KUKA KRL program: chk_w2_grp3_opn.src, chk_w2_grp3_opn.dat

--- chk_w2_grp3_opn.src ---
&ACCESS RV2
&REL 3
&COMMENT Check grampos Z3 abertos
&PARAM DISKPATH = Program/SubeRotine
&PARAM TEMPLATE = C:\KRC\Roboter\Template\vorgabe
&PARAM EDITMASK = *
DEF chk_w2_grp3_opn( )
;FOLD ; Programa de verificacao de grampos Z3 aberto;%{PE}%R 4.1.16,%MKUKATPBASIS,%CCOMMENT,%VNORMAL,%P 2:Programa de verificacao de grampos Z3 aberto
;ENDFOLD

$TIMER[10] = 0
$TIMER_STOP[10] = FALSE

;FOLD WAIT FOR ( IN 499 'Z1.1 ABERTO/ ACTROS Z3.1 OPN' );%{PE}%R 8.2.24,%MKUKATPBASIS,%CEXT_WAIT_FOR,%VEXT_WAIT_FOR,%P 2:, 4:, 5:$IN, 6:499, 7:Z1.1 ABERTO/ ACTROS Z3.1 OPN, 9:
WAIT FOR  ( $IN[499] )
;ENDFOLD
;FOLD WAIT FOR ( IN 505 'ACTROS Z3.2 OPN' );%{PE}%R 8.2.24,%MKUKATPBASIS,%CEXT_WAIT_FOR,%VEXT_WAIT_FOR,%P 2:, 4:, 5:$IN, 6:505, 7:ACTROS Z3.2 OPN, 9:
WAIT FOR  ( $IN[505] )
;ENDFOLD
;FOLD WAIT FOR ( IN 507 'ACTROS 3.3 OPN' );%{PE}%R 8.2.24,%MKUKATPBASIS,%CEXT_WAIT_FOR,%VEXT_WAIT_FOR,%P 2:, 4:, 5:$IN, 6:507, 7:ACTROS 3.3 OPN, 9:
WAIT FOR  ( $IN[507] )
;ENDFOLD
;FOLD WAIT FOR ( IN 509 'ACTROS 3.4 OPN' );%{PE}%R 8.2.24,%MKUKATPBASIS,%CEXT_WAIT_FOR,%VEXT_WAIT_FOR,%P 2:, 4:, 5:$IN, 6:509, 7:ACTROS 3.4 OPN, 9:
WAIT FOR  ( $IN[509] )
;ENDFOLD
;FOLD WAIT FOR ( IN 513 'Z3.2 ABERTO/ ACTROS Z3.5 OPN' );%{PE}%R 8.2.24,%MKUKATPBASIS,%CEXT_WAIT_FOR,%VEXT_WAIT_FOR,%P 2:, 4:, 5:$IN, 6:513, 7:Z3.2 ABERTO/ ACTROS Z3.5 OPN, 9:
WAIT FOR  ( $IN[513] )
;ENDFOLD
;FOLD WAIT FOR ( IN 515 'Z4.1 ABERTO/ ACTROS Z3.6 OPN' );%{PE}%R 8.2.24,%MKUKATPBASIS,%CEXT_WAIT_FOR,%VEXT_WAIT_FOR,%P 2:, 4:, 5:$IN, 6:515, 7:Z4.1 ABERTO/ ACTROS Z3.6 OPN, 9:
WAIT FOR  ( $IN[515] )
;ENDFOLD
;FOLD WAIT FOR ( NOT IN 500 'Z1.1 FECHADO/ ACTROS Z3.1 CLO' );%{PE}%R 8.2.24,%MKUKATPBASIS,%CEXT_WAIT_FOR,%VEXT_WAIT_FOR,%P 2:, 4:NOT, 5:$IN, 6:500, 7:Z1.1 FECHADO/ ACTROS Z3.1 CLO, 9:
WAIT FOR  (  NOT $IN[500] )
;ENDFOLD
;FOLD WAIT FOR ( NOT IN 506 'ACTROS 3.2 CLO' );%{PE}%R 8.2.24,%MKUKATPBASIS,%CEXT_WAIT_FOR,%VEXT_WAIT_FOR,%P 2:, 4:NOT, 5:$IN, 6:506, 7:ACTROS 3.2 CLO, 9:
WAIT FOR  (  NOT $IN[506] )
;ENDFOLD
;FOLD WAIT FOR ( NOT IN 508 'ACTROS 3.3 CLO' );%{PE}%R 8.2.24,%MKUKATPBASIS,%CEXT_WAIT_FOR,%VEXT_WAIT_FOR,%P 2:, 4:NOT, 5:$IN, 6:508, 7:ACTROS 3.3 CLO, 9:
WAIT FOR  (  NOT $IN[508] )
;ENDFOLD
;FOLD WAIT FOR NOT ( IN 510 'ACTROS 3.4 CLO' );%{PE}%R 8.2.24,%MKUKATPBASIS,%CEXT_WAIT_FOR,%VEXT_WAIT_FOR,%P 2:NOT, 4:, 5:$IN, 6:510, 7:ACTROS 3.4 CLO, 9:
WAIT FOR  NOT ( $IN[510] )
;ENDFOLD
;FOLD WAIT FOR ( NOT IN 514 'Z3.2 FECHADO/ ACTROS Z3.5 CLO' );%{PE}%R 8.2.24,%MKUKATPBASIS,%CEXT_WAIT_FOR,%VEXT_WAIT_FOR,%P 2:, 4:NOT, 5:$IN, 6:514, 7:Z3.2 FECHADO/ ACTROS Z3.5 CLO, 9:
WAIT FOR  (  NOT $IN[514] )
;ENDFOLD
;FOLD WAIT FOR ( NOT IN 516 'Z4.1 FECHADO/ ACTROS Z3.6 CLO' );%{PE}%R 8.2.24,%MKUKATPBASIS,%CEXT_WAIT_FOR,%VEXT_WAIT_FOR,%P 2:, 4:NOT, 5:$IN, 6:516, 7:Z4.1 FECHADO/ ACTROS Z3.6 CLO, 9:
WAIT FOR  (  NOT $IN[516] )
;ENDFOLD
$TIMER_STOP[10] = TRUE
$TIMER[10] = 0

END

--- chk_w2_grp3_opn.dat ---
&ACCESS RV2
&REL 3
&COMMENT Check grampos Z3 abertos
&PARAM DISKPATH = Program/SubeRotine
&PARAM TEMPLATE = C:\KRC\Roboter\Template\vorgabe
&PARAM EDITMASK = *
DEFDAT chk_w2_grp3_opn
;FOLD EXTERNAL DECLARATIONS;%{PE}%V3.2.0,%MKUKATPBASIS,%CEXT,%VCOMMON,%P
;FOLD BAS EXT;%{PE}%V3.2.0,%MKUKATPBASIS,%CEXT,%VEXT,%P
EXT  BAS (BAS_COMMAND  :IN,REAL  :IN )
DECL INT SUCCESS
;ENDFOLD
;FOLD GRIPPER EXT;%{E}%V3.2.0,%MKUKATPGRIPPER,%CEXT,%VEXT,%P
EXT  H50 (INT:IN, INT:IN ,INT:IN ,GRP_TYP:IN)
;ENDFOLD
;FOLD SPOT EXT;%{E}%V3.2.0,%MKUKATPSPOT,%CEXT,%VEXT,%P
EXT  USERSPOT (S_COMMAND  :IN, SPOT_TYPE:IN)
;ENDFOLD
;FOLD USER EXT;%{E}%V3.2.0,%MKUKATPUSER,%CEXT,%VEXT,%P
;Make here your modifications
;ENDFOLD
;ENDFOLD

ENDDAT
